TYPE LAxisCtrl_typePhasing :
STRUCT

	phaseShift               		: LREAL;
	velocity                 		: LREAL;
 	acceleration			: LREAL;
	deceleration			: LREAL;
	jerk                     			: LREAL;
	phaseAbsolute            		: BOOL;
	phaseShiftChangeOnTheFly 	: BOOL;

END_STRUCT
END_TYPE

(* stored: Version 1.1.0.1
   DUT LAxisCtrl_typePhasing: Id {d8ec1225-b341-4024-9764-2a30c603d207} *)
